PROGRAM MAIN
VAR
	
	//Pulsador AT %I*: BOOL;
	//Lampara AT %Q*: BOOL;
	
	Estacion: FB_Estacion;

END_VAR

Estacion();

END_PROGRAM

(* stored: Version 1.1.0.1, ProductVersion 3.1.4024.12
   POU MAIN: Id {e4a90306-f409-4a7b-93ef-0ed7f90ceaa4}, SpecialFunc None *)
